// TIA Portal V18 export
TYPE "LGasp_typeStampante"
// stored: IsFailsafeCompliant false
   STRUCT
      testostampa : WString[20];
      layoutStampa { ExternalAccessible := 'False'; ExternalVisible := 'False'; ExternalWritable := 'False'} : WString[20];
   END_STRUCT;
END_TYPE
